PROGRAM EVENTS
VAR
END_VAR

LogEvent_1000_1 (SourceID := 1000,EventID := 1,bSetEvent := bSetEvent_1000_1, bQuit := bQuitEvent_1000_1);
LogEvent_1000_2 (SourceID := 1000,EventID := 2,bSetEvent := bSetEvent_1000_2, bQuit := bQuitEvent_1000_2);

END_PROGRAM

(* stored: Version 1.1.0.1, ProductVersion 3.1.0.26
   POU EVENTS: Id {c85f5cf1-e497-4951-ada9-240704e86f60} *)
